FUNCTION_BLOCK MetalDosingOC (* CAT Function Block Type *)
  (* Standard: 61499-2 *)
  (* Version 0.0, 6/7/2026, Schneider Electric, template *)
  PACKAGE SE.Nereda;
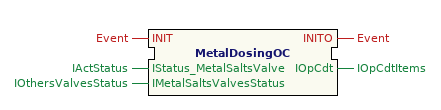
  EVENT_INPUT
    INIT;
  END_EVENT
  EVENT_OUTPUT
    INITO;
  END_EVENT
  SOCKETS
    IStatus_MetalSaltsValve : IActStatus;
    IMetalSaltsValvesStatus : IOthersValvesStatus;
  END_SOCKETS
  PLUGS
    IOpCdt : IOpCdtItems;
  END_PLUGS
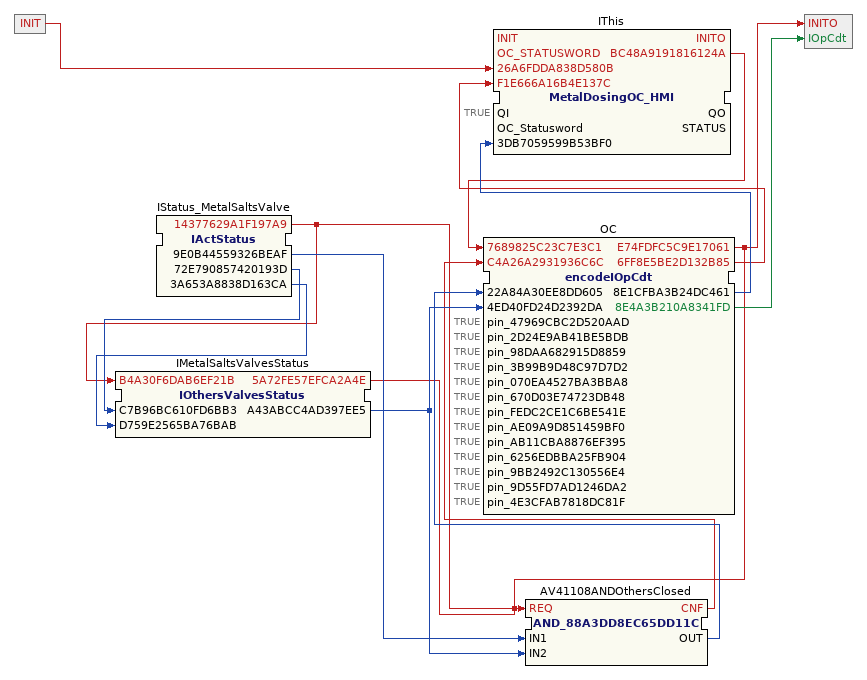
  (* 01 - FUNCTIONNAL INPUT INTERFACE *)
  (* 00 - INITIALIZATION *)
  (* 05 - LOGIC *)
  (* 06 - HMI INTERFACE *)
  (* 03 - FIELD INTERFACE *)
  (* Created by : Nouriddin OUECHEN 2026 *)
  (* Operating Condition Status *)
  (* Created by : Nouriddin OUECHEN 2026 *)
  (* 02 - FUNCTIONNAL OUTPUT INTERFACE *)
  (* Operating conditions : 1. Metal salts valve AV41108 is available and valves for other reactors (AV42108) are closed. 2. Metal salt dosing not active for another reactor. 3. No error from the metal salt dosing unit. *)
  (* Actuators Tags : - Feed valve :                                  AV4x101 - Lower level valve :                        AV4x102 - Air fill valve sludge discharge :    AV4x171 - Chemicals valve :                         AV4x108 - Discharge valve :                         AV4x103 - Vent aeration grid valve :             AV4x107 - Vent sludge grid valve :               AV4x172 *)
  FBS
    OC : encodeIOpCdt(pin_47969CBC2D520AAD := TRUE, pin_2D24E9AB41BE5BDB := TRUE, pin_98DAA682915D8859 := TRUE, pin_3B99B9D48C97D7D2 := TRUE, pin_070EA4527BA3BBA8 := TRUE, pin_670D03E74723DB48 := TRUE, pin_FEDC2CE1C6BE541E := TRUE, pin_AE09A9D851459BF0 := TRUE, pin_AB11CBA8876EF395 := TRUE, pin_6256EDBBA25FB904 := TRUE, pin_9BB2492C130556E4 := TRUE, pin_9D55FD7AD1246DA2 := TRUE, pin_4E3CFAB7818DC81F := TRUE); (* You set the operating conditions. For the inputs that are not used set a constant to TRUE. *)
    IThis : MetalDosingOC_HMI(QI := TRUE);
    AV41108ANDOthersClosed : AND_88A3DD8EC65DD11C; {SET_ATTRIBUTE(Configuration.GenericFBType.InterfaceParams, Runtime.Standard#CNT:=2;OUT:BOOL)}
  END_FBS
  EVENT_CONNECTIONS
    INIT TO IThis.26A6FDDA838D580B;
    IStatus_MetalSaltsValve.14377629A1F197A9 TO AV41108ANDOthersClosed.REQ;
    OC.E74FDFC5C9E17061 TO INITO;
    OC.6FF8E5BE2D132B85 TO IThis.F1E666A16B4E137C;
    IThis.BC48A9191816124A TO OC.7689825C23C7E3C1;
    OC.E74FDFC5C9E17061 TO AV41108ANDOthersClosed.REQ;
    AV41108ANDOthersClosed.CNF TO OC.C4A26A2931936C6C;
    IMetalSaltsValvesStatus.5A72FE57EFCA2A4E TO AV41108ANDOthersClosed.REQ;
    IStatus_MetalSaltsValve.14377629A1F197A9 TO IMetalSaltsValvesStatus.B4A30F6DAB6EF21B;
  END_CONNECTIONS
  DATA_CONNECTIONS
    OC.8E1CFBA3B24DC461 TO IThis.3DB7059599B53BF0;
    AV41108ANDOthersClosed.OUT TO OC.22A84A30EE8DD605;
    IStatus_MetalSaltsValve.9E0B44559326BEAF TO AV41108ANDOthersClosed.IN1;
    IMetalSaltsValvesStatus.A43ABCC4AD397EE5 TO AV41108ANDOthersClosed.IN2;
    IMetalSaltsValvesStatus.A43ABCC4AD397EE5 TO OC.4ED40FD24D2392DA;
    IStatus_MetalSaltsValve.72E790857420193D TO IMetalSaltsValvesStatus.C7B96BC610FD6BB3;
    IStatus_MetalSaltsValve.3A653A8838D163CA TO IMetalSaltsValvesStatus.D759E2565BA76BAB;
  END_CONNECTIONS
  ADAPTER_CONNECTIONS
    OC.8E4A3B210A8341FD TO IOpCdt;
  END_CONNECTIONS
END_FUNCTION_BLOCK
